//enum of mode of operations
{attribute 'strict'}
{attribute 'to_string'}
{attribute 'qualified_only'}
TYPE eWsl15_Modes:
(
	Segment:=		0,
	Run:=			1,
	Level:=			2,
	DimAndBLend:=	3,
	Gauge:=			4,
	Led:=			5,
	Demo:=			6
)USINT;
END_TYPE

(* stored: Version 1.1.0.1
   DUT eWsl15_Modes: Id {6f6b2195-a232-46b2-a356-b8ed535cb7ca} *)
